FUNCTION_BLOCK FB_CupSupplyModule
VAR_INPUT
	nLine						: INT;
	timerCheckCylinder_Up		: REAL := 10;
	timerCheckCylinder_Dw		: REAL := 10;
	timerCylinder_Up_extend		: REAL;
	timerCylinder_Suction		: REAL;
	timerCylinder_Suction_extend: REAL;
	timerCheckEmpty				: REAL := 10;
	timerCheckStuck				: REAL := 10;
	ttimerCylinder_val			: REAL;
	timerCylinder_Suction_pick	: REAL;
END_VAR
VAR_OUTPUT
END_VAR
VAR
	// ===== CHILD COMPONENTS ======
	fbCylinder_Up				: FB_Cylinder;
	fbCylinder_Dw				: FB_Cylinder;
	fbCylinder_Suction			: FB_Cylinder;
	// ===== SIM COMPONENTS ======
	fbCylinderSim_Up			: FB_Cylinder_Sim;
	fbCylinderSim_Dw			: FB_Cylinder_Sim;
	fbCylinderSim_Suction		: FB_Cylinder_Sim;
	// ===== INTERFACES ======
	iCylinder_Up				: I_Cylinder;
	iCylinder_Dw				: I_Cylinder;
	iCylinder_Suction			: I_Cylinder;
	//===== Var IO ======
	bCupEmpty AT %I*			: BOOL;
	bCupDrop  AT %I*			: BOOL;
	//===== Var Auto ====
	//===== Var method
	nState_DropCup				: INT;
	nState_Enable				: INT;
	nState_Check				: INT;
	nState_siren				: INT;
	nState_Reset				: INT;
	tTimer_Enable1				: TON;
	tTimer_Enable2				: TON;
	tTimer_DropCup				: TON;
	tTimer_CheckCup				: TON;
	tTimer_Suction				: TON;
	tTimer_Up					: ton;
	tTimer_Dw					: TON;
	tTimer_Reset				: TON;
END_VAR

IF bSimMode THEN
	iCylinder_Up := fbCylinderSim_Up;
	fbCylinderSim_Up();
	iCylinder_Dw := fbCylinderSim_Dw;
	fbCylinderSim_Dw();
	iCylinder_Suction := fbCylinderSim_Suction;
	fbCylinderSim_Suction();
ELSE
	iCylinder_Up := fbCylinder_Up;
	fbCylinder_Up(id := 1);
	iCylinder_Dw := fbCylinder_Dw;
	fbCylinder_Dw(id := 1);
	iCylinder_Suction := fbCylinder_Suction;
	fbCylinder_Suction(id := 1);
END_IF

METHOD CheckCup : BOOL
VAR_INPUT
END_VAR
IF NOT isCupEmpty THEN
	CASE nState_Check OF
		0:
			IF nLine = 1 THEN
				F_SetWarning(101,nLine := 1);
			ELSIF nLine = 2 THEN
				F_SetWarning(108,nLine := 2);
			END_IF
			nState_Check := 1;
		1: 
			tTimer_CheckCup(IN := TRUE, PT := REAL_TO_TIME(timerCheckEmpty)*1000);
			IF tTimer_CheckCup.Q THEN
				IF nLine = 1 THEN
						F_SetError(1,nLine := 1);
				ELSIF nLine = 2 THEN
						F_SetError(23,nLine := 2);
				END_IF
			END_IF
	END_CASE
ELSE
	tTimer_CheckCup(IN := FALSE);
	nState_Check := 0;
END_IF

CASE nState_siren OF
	0:
		IF NOT isCupEmpty THEN
			nState_siren := 1;
		END_IF
	1:
		IF isCupEmpty THEN
			IF nLine = 1 THEN
				bWrn := FALSE;
			ELSIF nLine = 2 THEN
				bWrn2 := FALSE;
			END_IF
			bSirens := FALSE;
			nState_siren := 0;
		END_IF
END_CASE
END_METHOD

METHOD DropCup : BOOL
VAR_INPUT
END_VAR
CASE nState_DropCup OF
	0: //init
		DropCup := FALSE;
		tTimer_DropCup(IN := FALSE);
		tTimer_Suction(IN := FALSE);
		nState_DropCup := 1;
	1: //check CupEmpty
		nState_DropCup := 2;
	2: //cylinder_up extend to hold cup
		iCylinder_Up.Extend();
		iCylinder_Suction.Retract();
		tTimer_Suction(IN := TRUE, PT := REAL_TO_TIME(timerCylinder_Suction_extend)*1000);
		tTimer_DropCup(IN := TRUE, PT := REAL_TO_TIME(timerCylinder_Up_extend)*1000);
		IF tTimer_DropCup.Q AND tTimer_Suction.Q THEN
			nState_DropCup := 3;
		END_IF
	3: // cylinder_dw retract to dropcup
		iCylinder_Up.Extend();
		tTimer_Suction(IN := FALSE);
		tTimer_DropCup(IN := FALSE);
		iCylinder_Dw.Retract();
		nState_DropCup := 33;
	33:
		iCylinder_Up.Extend();
		iCylinder_Dw.Retract();
		iCylinder_Suction.Retract();
		tTimer_DropCup(IN := TRUE, PT := REAL_TO_TIME(timerCheckCylinder_Dw)*1000);
		IF tTimer_DropCup.Q THEN
			IF nLine = 1 THEN
				F_SetError(4,nLine := 1);
			ELSIF nLine = 2 THEN
				F_SetError(26,nLine := 2);
			END_IF
		ELSIF iCylinder_Dw.bIsRetract THEN
			tTimer_DropCup(IN := FALSE);
			nState_DropCup := 34;
		END_IF
	34:
		tTimer_DropCup(IN := TRUE, PT := REAL_TO_TIME(timerCylinder_Suction_pick)*1000);
		IF tTimer_DropCup.Q THEN
			nState_DropCup := 44;
		END_IF
	44:
		tTimer_DropCup(IN := FALSE);
		nState_DropCup := 4;
	4: // check not isCupDrop
		iCylinder_Up.Extend();
		iCylinder_Dw.Retract();
		iCylinder_Suction.Extend();
		tTimer_Suction(IN := TRUE, PT := REAL_TO_TIME(timerCylinder_Suction)*1000);
		IF NOT isCupDrop THEN //sensor NC
			tTimer_DropCup(IN := FALSE);
			nState_DropCup := 5;
		ELSE
			tTimer_DropCup(IN := TRUE, PT := REAL_TO_TIME(timerCheckStuck)*1000);
			IF tTimer_DropCup.Q THEN
				IF nLine = 1 THEN
					F_SetError(2,nLine := 1);
					nState_DropCup := 5;
				ELSIF nLine = 2 THEN
					F_SetError(24,nLine := 2);
					nState_DropCup := 5;
				END_IF
			END_IF
		END_IF
	5:
		tTimer_Dw(IN := TRUE, PT := REAL_TO_TIME(ttimerCylinder_val)*1000);
		IF tTimer_Dw.Q THEN
			iCylinder_Dw.Extend();
		END_IF
		IF iCylinder_Suction.bIsExtend THEN
			tTimer_Suction(IN := FALSE);
			nState_DropCup := 55;
		ELSE
			tTimer_Suction(IN := TRUE, PT := REAL_TO_TIME(timerCylinder_Suction)*1000);
			IF tTimer_Suction.Q THEN
				IF nLine = 1 THEN
					F_SetError(60,nLine := 1);
				ELSIF nLine = 2 THEN
					F_SetError(61,nLine := 2);
				END_IF
			END_IF
		END_IF
	55:
		tTimer_Dw(IN := false);
		IF isCupDrop THEN
			tTimer_DropCup(IN := FALSE);
			nState_DropCup := 6;
		ELSE
			tTimer_DropCup(IN := TRUE, PT := REAL_TO_TIME(timerCheckStuck)*1000);
			IF tTimer_DropCup.Q  THEN
				IF nLine = 1 THEN
					F_SetError(2,nLine := 1);
				ELSIF nLine = 2 THEN
					F_SetError(24,nLine := 2);
				END_IF
			END_IF
		END_IF
	6: //complete
		iCylinder_Dw.Extend();
		tTimer_DropCup(IN := TRUE, PT := REAL_TO_TIME(timerCheckCylinder_Dw)*1000);
		IF tTimer_DropCup.Q THEN
			IF nLine = 1 THEN
				F_SetError(5,nLine := 1);
			ELSIF nLine = 2 THEN
				F_SetError(27,nLine := 2);
			END_IF
		ELSIF iCylinder_Dw.bIsExtend THEN
			tTimer_DropCup(IN := FALSE);
			nState_DropCup := 7;
		END_IF
	7:
		iCylinder_Up.Retract();
		tTimer_DropCup(IN := TRUE, PT := REAL_TO_TIME(timerCheckCylinder_Up)*1000);
		IF tTimer_DropCup.Q THEN
			IF nLine = 1 THEN
				F_SetError(3,nLine := 1);
			ELSIF nLine = 2 THEN
				F_SetError(25,nLine := 2);
			END_IF
		ELSIF iCylinder_Up.bIsRetract THEN
			DropCup := TRUE;
			tTimer_DropCup(IN := FALSE);
			nState_DropCup := 0;
		END_IF
END_CASE
END_METHOD

METHOD Enable : BOOL
VAR_INPUT
END_VAR
CASE nState_Enable OF
	0:
		Enable := FALSE;
		tTimer_Enable1(IN := FALSE);
		tTimer_Enable2(IN := FALSE);
		nState_Enable := 1;
	1:
		iCylinder_Up.Retract();
		iCylinder_Dw.Extend();
		nState_Enable := 2;
	2:
		tTimer_Enable1(IN := TRUE, PT := REAL_TO_TIME(timerCheckCylinder_Up));
		tTimer_Enable2(IN := TRUE, PT := REAL_TO_TIME(timerCheckCylinder_Dw));
		IF tTimer_Enable1.Q AND NOT iCylinder_Up.bIsRetract THEN
			IF nLine = 1 THEN
				F_SetError(3,nLine := 1);
				nState_Enable := 99;//error
			ELSIF nLine = 2 THEN
				F_SetError(21,nLine := 2);
				nState_Enable := 99;//error
			END_IF
		ELSIF tTimer_Enable2.Q AND NOT iCylinder_Dw.bIsExtend THEN
			IF nLine = 1 THEN
				F_SetError(4,nLine := 1);
				nState_Enable := 99;//error
			ELSIF nLine = 2 THEN
				F_SetError(22,nLine := 2);
				nState_Enable := 99;//error
			END_IF
		ELSIF iCylinder_Up.bIsRetract AND iCylinder_Dw.bIsExtend THEN
			tTimer_Enable1(IN := FALSE);
			tTimer_Enable2(IN := FALSE);
			nState_Enable := 3;
		END_IF
	3:
		Enable := TRUE;
	99://Error
END_CASE
END_METHOD

METHOD HoldCup : BOOL
VAR_INPUT
END_VAR
iCylinder_Up.Extend();
END_METHOD

METHOD Init : BOOL
VAR_INPUT
END_VAR
nState_DropCup				:= 0;
nState_Enable				:= 0;
END_METHOD

PROPERTY isCupDrop : BOOL
GET
isCupDrop := bCupDrop;
END_GET
END_PROPERTY

PROPERTY isCupEmpty : BOOL
GET
isCupEmpty := bCupEmpty;
END_GET
END_PROPERTY

METHOD Manual : BOOL
VAR_INPUT
	bCylinder_up_extend 			: BOOL;
	bCylinder_up_retract 			: BOOL;
	bCylinder_dw_extend 			: BOOL;
	bCylinder_dw_retract 			: BOOL;
	bCylinder_suction_extend 		: BOOL;
	bCylinder_suction_retract 		: BOOL;
END_VAR

VAR
	re: INT;
END_VAR
IF bCylinder_up_extend THEN
	iCylinder_Up.Extend();
END_IF

IF bCylinder_up_retract THEN
	iCylinder_Up.Retract();
	tTimer_Up(IN := TRUE, PT := REAL_TO_TIME(timerCheckCylinder_Up)*1000);
		IF tTimer_Up.Q THEN
			IF nLine = 1 THEN
				F_SetError(3,nLine := 1);
			ELSIF nLine = 2 THEN
				F_SetError(25,nLine := 2);
			END_IF
		ELSIF iCylinder_Up.bIsRetract THEN
			tTimer_Up(IN := FALSE);
		END_IF
END_IF

IF bCylinder_dw_extend THEN
	iCylinder_Dw.Extend();
	tTimer_Dw(IN := TRUE, PT := REAL_TO_TIME(timerCheckCylinder_Dw)*1000);
		IF tTimer_Dw.Q THEN
			IF nLine = 1 THEN
				F_SetError(5,nLine := 1);
			ELSIF nLine = 2 THEN
				F_SetError(27,nLine := 2);
			END_IF
		ELSIF iCylinder_Dw.bIsExtend THEN
			tTimer_Dw(IN := FALSE);
		END_IF;
END_IF

IF bCylinder_dw_retract THEN
	iCylinder_Dw.Retract();
	tTimer_Dw(IN := TRUE, PT := REAL_TO_TIME(timerCheckCylinder_Dw)*1000);
		IF tTimer_Dw.Q THEN
			IF nLine = 1 THEN
				F_SetError(4,nLine := 1);
			ELSIF nLine = 2 THEN
				F_SetError(26,nLine := 2);
			END_IF
		ELSIF iCylinder_Dw.bIsRetract THEN
			tTimer_Dw(IN := FALSE);
		END_IF;
END_IF

IF bCylinder_suction_retract THEN
	iCylinder_Suction.Retract();
END_IF

IF bCylinder_suction_extend THEN
	iCylinder_Suction.Extend();
	tTimer_Suction(IN := TRUE, PT := REAL_TO_TIME(timerCylinder_Suction)*1000);
		IF tTimer_Suction.Q THEN
			IF nLine = 1 THEN
				F_SetError(60,nLine := 1);
			ELSIF nLine = 2 THEN
				F_SetError(61,nLine := 2);
			END_IF
		ELSIF iCylinder_Suction.bIsExtend THEN
			tTimer_Suction(IN := FALSE);
		END_IF
END_IF
END_METHOD

METHOD Reset : BOOL
VAR_INPUT
END_VAR
tTimer_DropCup(IN := FALSE);
tTimer_Enable1(IN := FALSE);
tTimer_Enable2(IN := FALSE);
iCylinder_Suction.Extend();
tTimer_Up(IN := FALSE);
tTimer_Dw(IN := FALSE);
tTimer_Suction(IN := FALSE);
CASE nState_Reset OF
	0:
		tTimer_Reset(IN := TRUE, PT := T#300MS);
		iCylinder_Dw.Extend();
		IF tTimer_Reset.Q OR iCylinder_Dw.bIsExtend THEN
			nState_Reset := 1;
		END_IF
	1:
		tTimer_Reset(IN := FALSE);
		iCylinder_Up.Retract();
		nState_Reset := 0;
END_CASE
END_METHOD

METHOD Stop : BOOL
VAR_INPUT
END_VAR
tTimer_Enable1(IN := FALSE);
tTimer_Enable2(IN := FALSE);
tTimer_DropCup(IN := FALSE);
tTimer_Up(IN := FALSE);
tTimer_Dw(IN := FALSE);
tTimer_Suction(IN := false);
iCylinder_Dw.Extend();
END_METHOD

END_FUNCTION_BLOCK

(* stored: Version 1.1.0.1, ProductVersion 3.1.4024.12
   POU FB_CupSupplyModule: Id {230ce747-e2e8-43a7-b34c-18a5e1c3cba7}, SpecialFunc None
   Method CheckCup: Id {62e1e519-0717-476c-a1c1-ac14117a4a53}
   Method DropCup: Id {6774c00e-a692-4ec9-b43e-49a63117a206}
   Method Enable: Id {6071eec9-0c6b-4853-9e37-1c80cd49d6a5}
   Method HoldCup: Id {0941d1b1-8d35-4e8c-ba14-c0db4edf046a}
   Method Init: Id {c46dd9e3-de07-47e3-8476-52c0fc538db4}
   Property isCupDrop: Id {200df08e-2d70-4fe0-b116-65878b9d6ca0}
   Get Get: Id {ff92e2d5-e0ec-4b2e-b80d-885b1850e8f2}
   Property isCupEmpty: Id {748df038-ec64-4660-8ebb-a15b372a6204}
   Get Get: Id {2e67a479-5418-4f78-aa57-17ce7f227f91}
   Method Manual: Id {64ce3192-ada0-4203-a36b-e5948d3ff735}
   Method Reset: Id {dfc6ebf6-8e14-4982-9e12-11f6e5e8b417}
   Method Stop: Id {47c68cbb-60a2-4cd8-9a43-e4b7107cf7ff} *)
